// TIA Portal V20 export
DATA_BLOCK "BK15"   // DB301
// stored: MemoryReserve 100
   VAR
      "X10-1.CATHODE NG BOX FULL SENSOR" : Bool := FALSE;
      "X10-2.CATHODE NG BOX NG BOX DETECT SENSOR" : Bool := TRUE;
      "X12-1.CATHODE NG BOX LIFT DOWN" : Bool := FALSE;
      "X12-2.CATHODE NG BOX LIFT UP" : Bool := TRUE;
      "X14-1.CATHODE NG BOX LOCK DOWN" : Bool := TRUE;
      "X14-2.CATHODE NG BOX LOCK UP" : Bool := FALSE;
      "X16-1.SPARE" : Bool := FALSE;
      "X16-2.SPARE" : Bool := FALSE;
   END_VAR
BEGIN
END_DATA_BLOCK
